TYPE ST_SectionBase :
STRUCT
	SectionID 	: UINT;
	SectionLen	: UDINT;
END_STRUCT
END_TYPE

(* stored: Version 1.1.0.1, ProductVersion 3.1.4024.12
   DUT ST_SectionBase: Id {3a979e12-dc77-4c44-9fc6-ab044ac6092f} *)
